{attribute addProperty BoxType "EL3151-0000-0016"}
{attribute addProperty Id "AI_StandardAT %I*AI_Standard_8749C235749.250WcStateAT %I*WcState_98A4DF7520.250InfoDataAT %I*InfoData_BC63D37F80100"}
{attribute addProperty CRC "2717975163"}
{attribute addProperty SizeInBites "156"}
{attribute addProperty SizeInBytes "19.5"}
TYPE EL3151_32A64D67 :
STRUCT
	{attribute addProperty Name "AI_Standard"}
	AI_Standard : AI_Standard_8749C235;
	{attribute addProperty Name "WcState"}
	WcState : WcState_98A4DF75;
	{attribute addProperty Name "InfoData"}
	InfoData : InfoData_BC63D37F;
END_STRUCT
END_TYPE

(* stored: Version 1.2.0.0, ProductVersion 3.1.4024.9
   DUT EL3151_32A64D67: Id {3a6f5e5d-f064-43a9-aeda-f13675396d95} *)
